PROGRAM LimitSwitches
VAR
	StopMotorA : MC_Stop;
	StopMotorB : MC_Stop;
	ResetMotorA : MC_Reset;
	ResetMotorB : MC_Reset;
	
	casestate : INT;
END_VAR

CASE  casestate  OF 
	0 : //initialisation. If Axis is ready, then prepare to hit limit switch, if not, do nothing
	IF  PrepareAxes.switchcase = Implicit_Enum__PrepareAxes__switchcase.Movement THEN 
		casestate := 10;
		ELSE 
			//chill here
	END_IF
	10 : // Check If Limit Switch Triggered 
	IF GVL.LimitSwitchBotLeft OR GVL.LimitSwitchBotRight OR GVL.LimitSwitchMidLeft OR GVL.LimitSwitchMidRight OR GVL.LimitSwitchTopLeft OR GVL.LimitSwitchTopRight THEN 
		 StopMotorA(Execute := TRUE, Axis:= GVL.StepperReferenceA) ;  (* actual function to stop the motor *)
		 StopMotorB(Execute := TRUE,Axis:= GVL.StepperReferenceB) ;  (* actual function to stop the motor *)
		 casestate := 20; 
		 ELSE 
		ResetMotorA (Execute := FALSE, Axis := GVL.StepperReferenceA); (*Reset the Motors *)
		ResetMotorB (Execute := FALSE, Axis := GVL.StepperReferenceB); (*Reset the Motors *)
			 //chill again. Wait for Lim Switch Activation 
	END_IF
	
	20 : // Wait for Limit Switches to NOT be pressed before allowing movement again
	IF GVL.LimitSwitchBotLeft = FALSE AND GVL.LimitSwitchBotRight = FALSE AND GVL.LimitSwitchMidLeft = FALSE AND GVL.LimitSwitchMidRight = FALSE AND GVL.LimitSwitchTopLeft = FALSE AND GVL.LimitSwitchTopRight = FALSE THEN 
		casestate := 30 ;
		ELSE 
			//chill	
	END_IF
			
	30 : 
		
		IF StopMotorA.Active = FALSE THEN // IF FB not active, stop and start the FB 
		StopMotorA(Execute := TRUE, Axis:= GVL.StepperReferenceA) ;  (* actual function to stop the motor *)
		StopMotorB(Execute := TRUE,Axis:= GVL.StepperReferenceB) ;  (* actual function to stop the motor *)
		casestate := 40; 
		ELSIF StopMotorA.Active = TRUE THEN  //After Stopping and Starting, If ACtive = True continue as per normal
		ResetMotorA (Execute := TRUE, Axis := GVL.StepperReferenceA); (*Reset the Motors *)
		ResetMotorB (Execute := TRUE, Axis := GVL.StepperReferenceB); (*Reset the Motors *)
		StopMotorA(Execute := FALSE, Axis:= GVL.StepperReferenceA) ;  (* actual function to continue the motor *)
		StopMotorB(Execute := FALSE,Axis:= GVL.StepperReferenceB) ;  (* actual function to continue the motor *)
		casestate := 0;
		END_IF
	40 :  // Buffer for resetting the FB 
		casestate := 30;
		
END_CASE

END_PROGRAM

(* stored: Version 1.1.0.1, ProductVersion 3.1.4024.12
   POU LimitSwitches: Id {6ecd7bb5-2a35-46c9-88f2-7b7269e77e8a}, SpecialFunc None *)
